% RSLogix 500 project PROJECT 1  CGT PART 3.RSS, saved by version 8.30.00.16 %
PROJECT "P1_PJ3"    % processor: Bul.1763 MicroLogix 1100 Series B %

PROGRAM FILES
  LAD 2 "SECTIONS"  4 rungs
  LAD 3 "LOGIC"  16 rungs
  LAD 4 "INPUT"  3 rungs
  LAD 5 "OUTPUT"  3 rungs

DATA FILES
  O0 OUTPUT  4 elements
  I1 INPUT  6 elements
  S2 STATUS  66 elements
  B3 BINARY  1 elements
  T4 TIMER  2 elements
  C5 COUNTER  1 elements
  R6 CONTROL  1 elements
  N7 INTEGER  1 elements
  F8 FLOAT  1 elements

LADDER 2 "SECTIONS"
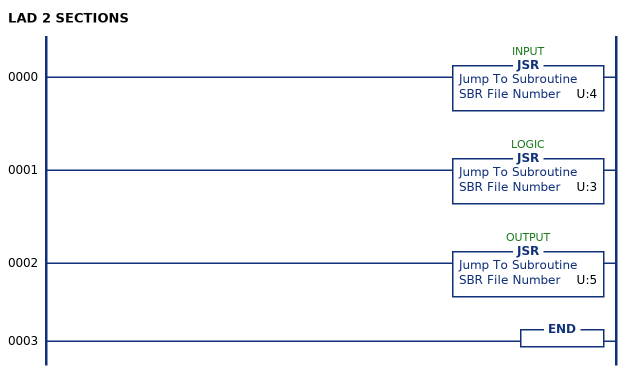
% Rung: 0 %  % edit flag set %
SOR JSR U:4 EOR
%   U:4  "INPUT" %
% Rung: 1 %  % edit flag set %
SOR JSR U:3 EOR
%   U:3  "LOGIC" %
% Rung: 2 %  % edit flag set %
SOR JSR U:5 EOR
%   U:5  "OUTPUT" %
% Rung: 3 %
SOR END EOR

LADDER 3 "LOGIC"
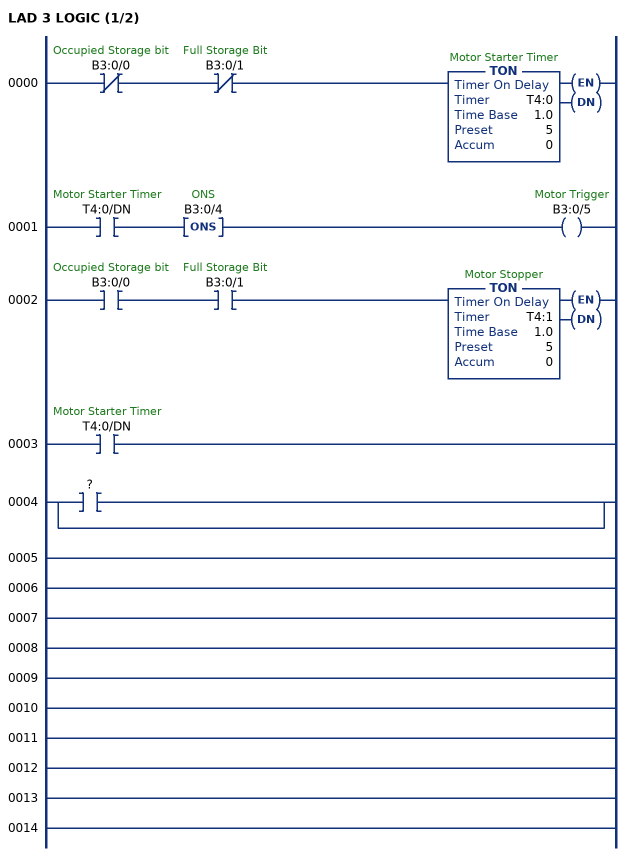
% Rung: 0 %
SOR XIO B3:0/0 XIO B3:0/1 TON T4:0 1.0 5 0 EOR
%   B3:0/0  "Occupied Storage bit" %
%   B3:0/1  "Full Storage Bit" %
%   T4:0  "Motor Starter Timer" %
% Rung: 1 %
SOR XIC T4:0/DN ONS B3:0/4 OTE B3:0/5 EOR
%   T4:0  "Motor Starter Timer" %
%   B3:0/4  "ONS" %
%   B3:0/5  "Motor Trigger" %
% Rung: 2 %
SOR XIC B3:0/0 XIC B3:0/1 TON T4:1 1.0 5 0 EOR
%   B3:0/0  "Occupied Storage bit" %
%   B3:0/1  "Full Storage Bit" %
%   T4:1  "Motor Stopper" %
% Rung: 3 %  % edit flag set %
SOR XIC T4:0/DN EOR
%   T4:0  "Motor Starter Timer" %
% Rung: 4 %  % edit flag set %
SOR BST XIC ? NXB BND EOR
% Rung: 5 %  % edit flag set %
SOR EOR
% Rung: 6 %  % edit flag set %
SOR EOR
% Rung: 7 %  % edit flag set %
SOR EOR
% Rung: 8 %  % edit flag set %
SOR EOR
% Rung: 9 %  % edit flag set %
SOR EOR
% Rung: 10 %  % edit flag set %
SOR EOR
% Rung: 11 %  % edit flag set %
SOR EOR
% Rung: 12 %  % edit flag set %
SOR EOR
% Rung: 13 %  % edit flag set %
SOR EOR
% Rung: 14 %  % edit flag set %
SOR EOR

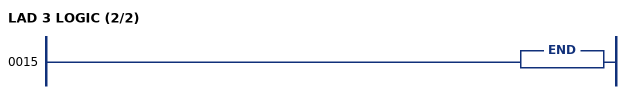
% Rung: 15 %
SOR END EOR

LADDER 4 "INPUT"
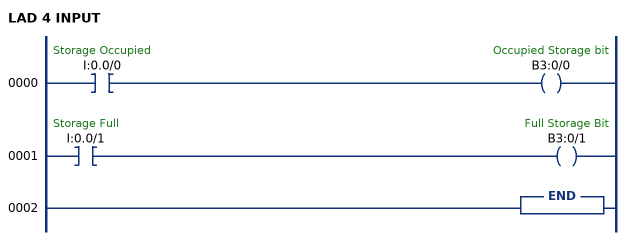
% Rung: 0 %
SOR XIC I:0.0/0 OTE B3:0/0 EOR
%   I:0.0/0  "Storage Occupied" %
%   B3:0/0  "Occupied Storage bit" %
% Rung: 1 %
SOR XIC I:0.0/1 OTE B3:0/1 EOR
%   I:0.0/1  "Storage Full" %
%   B3:0/1  "Full Storage Bit" %
% Rung: 2 %
SOR END EOR

LADDER 5 "OUTPUT"
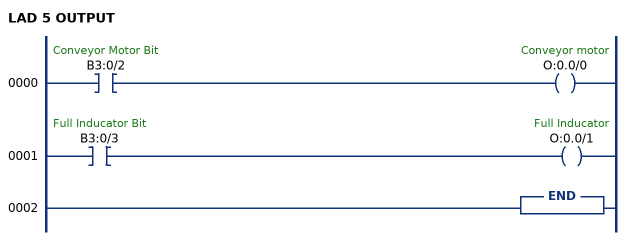
% Rung: 0 %
SOR XIC B3:0/2 OTE O:0.0/0 EOR
%   B3:0/2  "Conveyor Motor Bit" %
%   O:0.0/0  "Conveyor motor" %
% Rung: 1 %
SOR XIC B3:0/3 OTE O:0.0/1 EOR
%   B3:0/3  "Full Inducator Bit" %
%   O:0.0/1  "Full Inducator" %
% Rung: 2 %
SOR END EOR

DATA TABLE (non-zero values as saved)
DATA T4
% .PRE .ACC %
% T4:0 % 5 0
% T4:1 % 5 0
